{attribute 'GeneratedUsingTerminal: EL7201-0001-0017'}
{attribute addProperty BoxType "EL7201-0001-0017"}
{attribute addProperty Id "Position_actual_valueAT %I*UDINT4"}
{attribute addProperty CRC "131878004"}
{attribute addProperty Size "4"}
TYPE DS402_Position_actual_value_07DC4C74 EXTENDS InputBase_8311D824 :
STRUCT
	{attribute addProperty Name "Position_actual_value"}
	Position_actual_value AT %I* : UDINT;
END_STRUCT
END_TYPE

(* stored: Version 1.2.0.0, ProductVersion 3.1.4024.11
   DUT DS402_Position_actual_value_07DC4C74: Id {73cb179f-d2a9-4cfc-990d-64cf00655189} *)
